// TwinCAT 3 PLC project Untitled1
// ProgramVersion: 3.1.4024.0
// libraries:
//   Tc2_Standard, * (Beckhoff Automation GmbH)
//   Tc2_System, * (Beckhoff Automation GmbH)
//   Tc3_Module, * (Beckhoff Automation GmbH)
// project tree:
//   / PlcTask.TcTTO
//   POUs/ FB_ErrorManager.TcPOU, MAIN.TcPOU, ST_Error.TcDUT
// real-time tasks:
//   TASK PlcTask: cycle T#10ms, priority 20, ADS port 350

CONFIGURATION Untitled1
    RESOURCE PLC ON TwinCAT3
        TASK PlcTask(INTERVAL := T#10ms, PRIORITY := 20);
        PROGRAM MAIN WITH PlcTask : MAIN;
    END_RESOURCE
END_CONFIGURATION

// ---- POUs/ST_Error.TcDUT
TYPE ST_Error :
STRUCT
	ErrorMessage : STRING;
	ErrorCode : UINT;
END_STRUCT
END_TYPE

// ---- POUs/MAIN.TcPOU
PROGRAM MAIN
VAR
	fbErrorManager : FB_ErrorManager;
	bClear: BOOL;
	bError: BOOL;
	ErrorCode: UINT;
	ErrorMsg: STRING;
END_VAR

IF bClear THEN
	fbErrorManager.ClearError();
	bClear := FALSE;
END_IF

IF bError THEN
	bError := FALSE;
	fbErrorManager.RaiseError(ErrorCode, ErrorMsg);
END_IF

END_PROGRAM

// ---- POUs/FB_ErrorManager.TcPOU
FUNCTION_BLOCK FB_ErrorManager
VAR
	ErrorList : ARRAY[0..20] OF ST_Error;
	index : INT;
END_VAR

METHOD ClearError : BOOL
VAR_INPUT
END_VAR
index := 0;
MEMSET(ADR(ErrorList), 0, SIZEOF(ErrorList));
END_METHOD

METHOD RaiseError : BOOL
VAR_INPUT
	ErrorCode : UINT;
	ErrorMsg : STRING;
END_VAR
VAR
	i : INT;
END_VAR
IF index < 0 OR index >= 20 THEN
	RaiseError := FALSE;
	RETURN;
END_IF

FOR i := 0 TO 20 BY 1 DO
	IF ErrorList[i].ErrorCode = ErrorCode THEN
		RaiseError := FALSE;
		RETURN;
	END_IF
END_FOR

ErrorList[index].ErrorCode := ErrorCode;
ErrorList[index].ErrorMessage := ErrorMsg;
index := index + 1;
RaiseError := TRUE;
END_METHOD

END_FUNCTION_BLOCK
